VAR_GLOBAL
	
	AOUT AT %Q*	:	ARRAY[1..8] OF INT;
	
	XMEAS:	ARRAY[1..41] OF LREAL;
	MBS_XMEAS:	ARRAY[1..2] OF REAL;
	
END_VAR

(* stored: Version 1.1.0.1, ProductVersion 3.1.0.36
   GVL G_IO: Id {5c9be23e-5154-4405-95ca-9dd299cf237d} *)
